(* IEC 61131-3 sources: TSA-FMICS22/ahorn/test/lib_sa/file, 5 files *)

(* ---- field_access_of_callee.st ---- *)
PROGRAM P
VAR_INPUT
    a : INT;
END_VAR
VAR
    f : Fb;
END_VAR
VAR
    b : BOOL;
END_VAR
VAR_OUTPUT
    c : BOOL;
END_VAR
    f(x:=a,z=>b);
    IF f.z THEN
        c := TRUE;
    ELSE
        c := FALSE;
    END_IF;
END_PROGRAM

FUNCTION_BLOCK Fb
VAR_INPUT
    x : INT;
END_VAR
VAR
    y : INT;
END_VAR
VAR_OUTPUT
    z : BOOL;
END_VAR;
    IF x >= 32 THEN
        y := y;
    ELSE
        y := y + 1;
    END_IF;
    IF y >= 3 THEN
        z := TRUE;
    ELSE
        z := FALSE;
    END_IF;
END_FUNCTION_BLOCK

(* ---- modified_antivalent.st ---- *)
PROGRAM SFAntivalent2
VAR_INPUT
    Activate           : BOOL;
    SChannelNC         : SAFEBOOL;
    SChannelNO         : SAFEBOOL;
    DiscrepancyTime    : TIME;
END_VAR
VAR
    T1 : TONX;
    T1ET : TIME;
    T1Q : BOOL;
END_VAR
VAR_OUTPUT
    Ready              : BOOL;
    SAntivalentOut     : BOOL;
    Error              : BOOL;
    DiagCode           : WORD;
END_VAR

IF NOT Activate THEN
    DiagCode := 16#0000;
ELSE

CASE DiagCode OF
16#0000:
    IF Activate THEN
        DiagCode := 16#8001;
    END_IF;
16#8001:
    IF SChannelNC AND SChannelNO THEN
        DiagCode := 16#8004;
        T1(IN:=TRUE, PT:=DiscrepancyTime, ET=>T1ET, Q=>T1Q);
    ELSIF NOT SChannelNC AND NOT SChannelNO THEN
        DiagCode := 16#8014;
        T1(IN:=TRUE, PT:=DiscrepancyTime, ET=>T1ET, Q=>T1Q);
    ELSIF SChannelNC AND NOT SChannelNO THEN
        DiagCode := 16#8000;
    END_IF;
16#8004:
    IF T1Q THEN
        DiagCode := 16#C001;
    ELSIF NOT SChannelNC THEN
        DiagCode := 16#8001;
    ELSIF NOT SChannelNO THEN
        DiagCode := 16#8000;
    END_IF;
16#C001,
16#C002:
    IF NOT SChannelNC AND SChannelNO THEN
        DiagCode := 16#8001;
    END_IF;
16#8014:
    IF T1Q THEN
        DiagCode := 16#C002;
    ELSIF SChannelNO THEN
        DiagCode := 16#8001;
    ELSIF SChannelNC THEN
        DiagCode := 16#8000;
    END_IF;
16#C003:
    IF NOT SChannelNC AND SChannelNO THEN
        DiagCode := 16#8001;
    END_IF;
16#8005:
    IF T1Q THEN
        DiagCode := 16#C003;
    ELSIF NOT SChannelNC AND SChannelNO THEN
        DiagCode := 16#8001;
    END_IF;
16#8000:
    IF NOT SChannelNC OR SChannelNO THEN
        DiagCode := 16#8005;
        T1(IN:=TRUE, PT:=DiscrepancyTime, ET=>T1ET, Q=>T1Q);
    ELSIF NOT SChannelNC AND SChannelNO THEN
        DiagCode := 16#8001;
    END_IF;
END_CASE;
END_IF;

CASE DiagCode OF
16#0000:
    T1(IN:=FALSE, PT:=DiscrepancyTime, ET=>T1ET, Q=>T1Q);
    Ready := FALSE;
    Error := FALSE;
    SAntivalentOut:= FALSE;
16#8000:
    T1(IN:=FALSE, PT:=DiscrepancyTime, ET=>T1ET, Q=>T1Q);
    Ready := TRUE;
    Error := FALSE;
    SAntivalentOut := TRUE;
16#8001:
    T1(IN:=FALSE, PT:=DiscrepancyTime, ET=>T1ET, Q=>T1Q);
    Ready := TRUE;
    Error := FALSE;
    SAntivalentOut:= FALSE;
16#8004,
16#8014,
16#8005:
	T1(IN:=TRUE, PT:=DiscrepancyTime, ET=>T1ET, Q=>T1Q);
    Ready := TRUE;
    Error := FALSE;
    SAntivalentOut:= FALSE;
16#C001,
16#C002,
16#C003:
    T1(IN:=FALSE, PT:=DiscrepancyTime, ET=>T1ET, Q=>T1Q);
    Ready := TRUE;
    Error := TRUE;
    SAntivalentOut:= FALSE;
END_CASE;

END_PROGRAM

FUNCTION_BLOCK TONX
VAR_INPUT
  IN : BOOL;
  PT : TIME;
END_VAR
VAR
  running : BOOL;
END_VAR
VAR_TEMP
    timeout : BOOL;
END_VAR
VAR_OUTPUT
  Q : BOOL;
  ET : TIME;
END_VAR

  timeout := NONDETERMINISTIC_BOOL();

  IF NOT IN THEN
    Q := FALSE;
    running := FALSE;
  ELSIF NOT running AND NOT Q THEN
    running := TRUE;
  ELSIF running AND NOT Q THEN
    Q := timeout;
    running := NOT Q;
  END_IF;

  ET := NONDETERMINISTIC_TIME();
END_FUNCTION_BLOCK

(* ---- unreachable_branch_in_call.st ---- *)
PROGRAM P
VAR_INPUT
    a : INT;
END_VAR
VAR
    f : Fb;
END_VAR
VAR_OUTPUT
    b : BOOL;
END_VAR
    f(x:=a,z=>b);
END_PROGRAM

FUNCTION_BLOCK Fb
VAR_INPUT
    x : INT;
END_VAR
VAR
    y : INT;
END_VAR
VAR_OUTPUT
    z : BOOL;
END_VAR;
    IF x >= 32 THEN
        y := y + 1;
    ELSE
        y := y;
    END_IF;
    IF FALSE THEN
        z := TRUE;
        y := 0;
    ELSE
        z := FALSE;
    END_IF;
END_FUNCTION_BLOCK

(* ---- unreachable_branch_realizable_path.st ---- *)
PROGRAM P
VAR_INPUT
    a : INT;
END_VAR
VAR
    f : Fb;
END_VAR
VAR
    b : BOOL;
END_VAR
VAR_OUTPUT
    c : BOOL;
END_VAR
    IF a >= 32 THEN
        f(x:=a,z=>b);
        IF b THEN
            c := TRUE;
        ELSE
            c := FALSE;
        END_IF;
    ELSE
        f(x:=a,z=>b);
    END_IF;
END_PROGRAM

FUNCTION_BLOCK Fb
VAR_INPUT
    x : INT;
END_VAR
VAR_OUTPUT
    z : BOOL;
END_VAR;
    IF x < 32 THEN
        z := TRUE;
    ELSE
        z := FALSE;
    END_IF;
END_FUNCTION_BLOCK

(* ---- unreachable_branches_of_antivalent.st ---- *)
PROGRAM P
VAR_INPUT
    Activate       : BOOL := FALSE;
END_VAR
VAR
    Ready          : BOOL := FALSE;
    STwoHandOut   : BOOL := FALSE;
    DiagCode       : WORD := 16#0;
END_VAR
    IF NOT Activate THEN
        DiagCode := 16#0000;
    ELSE
     CASE DiagCode OF
     16#0000:
         IF Activate THEN
              DiagCode := 16#8001;
         END_IF;
     END_CASE;
    END_IF;

    CASE DiagCode OF
    16#0000:
        Ready := FALSE;
        STwoHandOut := FALSE;
    16#8000:
        Ready := TRUE;
        STwoHandOut := TRUE;
    16#8001:
        Ready := TRUE;
        STwoHandOut := FALSE;
    END_CASE;
END_PROGRAM
